(* Schneider Machine Expert - Basic project Pump_Tank_Backup_System_IL, file version 3.0.0.0 *)

HARDWARE
  EthernetConfiguration: SubnetMask=255.255.255.0
  SerialLineConfiguration: Parity=Even, DataBits=8, StopBits=1

SYMBOLS  (address, symbol, comment, settings)
  %TM0      PUMP1_START_DELAY  "Pump 1 Startup Delay - 2 seconds before speed check"  [Type=TON, TimeBase=TimeBase1s, Preset=2]
  %TM1      PUMP2_START_DELAY  "Pump 2 Startup Delay - 2 seconds before speed check"  [Type=TON, TimeBase=TimeBase1s, Preset=2]
  %TM2      PUMP3_START_DELAY  "Pump 3 Startup Delay - 2 seconds before speed check"  [Type=TON, TimeBase=TimeBase1s, Preset=2]
  %I0.0     START_BTN  "System Start Button"
  %I0.1     STOP_BTN  "System Stop Button (NC)"
  %I0.2     E_STOP  "Emergency Stop (NC)"
  %I0.3     PUMP1_SPEED_OK  "Pump 1 Zero Speed Sensor (NC)"
  %I0.4     PUMP2_SPEED_OK  "Pump 2 Zero Speed Sensor (NC)"
  %I0.5     PUMP3_SPEED_OK  "Pump 3 Zero Speed Sensor (NC)"
  %I0.6     TANK1_LOW  "Tank 1 Low Level Switch"
  %I0.7     TANK1_HIGH  "Tank 1 High Level Switch"
  %I0.8     TANK2_LOW  "Tank 2 Low Level Switch"
  %I0.9     TANK2_HIGH  "Tank 2 High Level Switch"
  %I0.10    TANK3_LOW  "Tank 3 Low Level Switch"
  %I0.11    TANK3_HIGH  "Tank 3 High Level Switch"
  %I0.12    PUMP1_OL  "Pump 1 Overload (NC)"
  %I0.13    PUMP2_OL  "Pump 2 Overload (NC)"
  %I0.14    PUMP3_OL  "Pump 3 Overload (NC)"
  %I0.15    FAULT_RESET  "Fault Reset Button"
  %Q0.0     PUMP1_RUN  "Pump 1 Motor Contactor"
  %Q0.1     PUMP2_RUN  "Pump 2 Motor Contactor"
  %Q0.2     PUMP3_RUN  "Pump 3 Motor Contactor"
  %Q0.3     VALVE_12  "Valve Between Tank 1-2"
  %Q0.4     VALVE_23  "Valve Between Tank 2-3"
  %Q0.5     VALVE_13  "Valve Between Tank 1-3"
  %Q0.6     PUMP1_FAULT_IND  "Pump 1 Fault Indicator"
  %Q0.7     PUMP2_FAULT_IND  "Pump 2 Fault Indicator"
  %Q0.8     PUMP3_FAULT_IND  "Pump 3 Fault Indicator"
  %Q0.9     SYSTEM_RUN_IND  "System Running Indicator"
  %Q0.10    ALARM_OUTPUT  "General Alarm Horn"
  %M0       SYSTEM_RUN  "System Running Flag"
  %M1       PUMP1_CMD  "Pump 1 Command"
  %M2       PUMP2_CMD  "Pump 2 Command"
  %M3       PUMP3_CMD  "Pump 3 Command"
  %M10      PUMP1_FAULT  "Pump 1 Fault (Latched)"
  %M11      PUMP2_FAULT  "Pump 2 Fault (Latched)"
  %M12      PUMP3_FAULT  "Pump 3 Fault (Latched)"
  %M20      TANK1_NEEDS_BACKUP  "Tank 1 Backup Mode"
  %M21      TANK2_NEEDS_BACKUP  "Tank 2 Backup Mode"

PouDescriptor Pump_Tank_Backup_IL_Main
  (* PouType=Program *)

// Rung 0: Rung 1
// System Start/Stop with Emergency Stop - Seal-in Circuit
  LD %I0.0                (* START_BTN - Load START button *)
  OR %M0                  (* SYSTEM_RUN - OR with SYSTEM_RUN (seal-in) *)
  ANDN %I0.1              (* STOP_BTN - AND NOT STOP button (NC) *)
  ANDN %I0.2              (* E_STOP - AND NOT E_STOP (NC) *)
  ST %M0                  (* SYSTEM_RUN - Store to SYSTEM_RUN flag *)
  // as ST:
  //   SYSTEM_RUN := (START_BTN OR SYSTEM_RUN) AND NOT STOP_BTN AND NOT E_STOP;

// Rung 1: Rung 2
// Pump 1 Command - Fill Tank 1 when low, stop at high
  LD %M0                  (* SYSTEM_RUN - System running *)
  AND %I0.6               (* TANK1_LOW - AND Tank 1 low level *)
  ANDN %I0.7              (* TANK1_HIGH - AND NOT Tank 1 high level *)
  ANDN %M10               (* PUMP1_FAULT - AND NOT Pump 1 fault *)
  ANDN %I0.12             (* PUMP1_OL - AND NOT Pump 1 overload *)
  ST %M1                  (* PUMP1_CMD - Store to PUMP1_CMD *)
  // as ST:
  //   PUMP1_CMD := SYSTEM_RUN AND TANK1_LOW AND NOT TANK1_HIGH AND NOT PUMP1_FAULT AND NOT PUMP1_OL;

// Rung 2: Rung 3
// Pump 2 Command - Fill Tank 2 when low, stop at high
  LD %M0                  (* SYSTEM_RUN - System running *)
  AND %I0.8               (* TANK2_LOW - AND Tank 2 low level *)
  ANDN %I0.9              (* TANK2_HIGH - AND NOT Tank 2 high level *)
  ANDN %M11               (* PUMP2_FAULT - AND NOT Pump 2 fault *)
  ANDN %I0.13             (* PUMP2_OL - AND NOT Pump 2 overload *)
  ST %M2                  (* PUMP2_CMD - Store to PUMP2_CMD *)
  // as ST:
  //   PUMP2_CMD := SYSTEM_RUN AND TANK2_LOW AND NOT TANK2_HIGH AND NOT PUMP2_FAULT AND NOT PUMP2_OL;

// Rung 3: Rung 4
// Pump 3 Command - Fill Tank 3 when low, stop at high
  LD %M0                  (* SYSTEM_RUN - System running *)
  AND %I0.10              (* TANK3_LOW - AND Tank 3 low level *)
  ANDN %I0.11             (* TANK3_HIGH - AND NOT Tank 3 high level *)
  ANDN %M12               (* PUMP3_FAULT - AND NOT Pump 3 fault *)
  ANDN %I0.14             (* PUMP3_OL - AND NOT Pump 3 overload *)
  ST %M3                  (* PUMP3_CMD - Store to PUMP3_CMD *)
  // as ST:
  //   PUMP3_CMD := SYSTEM_RUN AND TANK3_LOW AND NOT TANK3_HIGH AND NOT PUMP3_FAULT AND NOT PUMP3_OL;

// Rung 4: Rung 5
// Pump 1 Startup Timer and Motor Output
  BLK %TM0                (* PUMP1_START_DELAY - Begin Timer 0 block (PUMP1_START_DELAY) *)
  LD %M1                  (* PUMP1_CMD - Load Pump 1 command *)
  IN                      (* Timer input - starts 2s delay *)
  END_BLK                 (* End timer block *)
  LD %M1                  (* PUMP1_CMD - Load Pump 1 command *)
  ST %Q0.0                (* PUMP1_RUN - Output to PUMP1_RUN contactor *)
  // as ST:
  //   PUMP1_START_DELAY(IN := PUMP1_CMD);
  //   PUMP1_RUN := PUMP1_CMD;

// Rung 5: Rung 6
// Pump 1 Zero Speed Fault - Latching with Reset
  LD %TM0.Q               (* PUMP1_START_DELAY - Timer done (2s elapsed) *)
  ANDN %I0.3              (* PUMP1_SPEED_OK - AND NOT speed OK (zero speed detected) *)
  OR %M10                 (* PUMP1_FAULT - OR with fault latch (seal-in) *)
  ANDN %I0.15             (* FAULT_RESET - AND NOT fault reset button *)
  ST %M10                 (* PUMP1_FAULT - Store to PUMP1_FAULT (latched) *)
  // as ST:
  //   PUMP1_FAULT := (PUMP1_START_DELAY.Q AND NOT PUMP1_SPEED_OK OR PUMP1_FAULT) AND NOT FAULT_RESET;

// Rung 6: Rung 7
// Pump 2 Output - Normal Operation or Backup for Tank 1
  BLK %TM1                (* PUMP2_START_DELAY - Begin Timer 1 block (PUMP2_START_DELAY) *)
  LD %M2                  (* PUMP2_CMD - Load Pump 2 command *)
  OR %M20                 (* TANK1_NEEDS_BACKUP - OR Tank 1 needs backup *)
  IN                      (* Timer input *)
  END_BLK                 (* End timer block *)
  LD %M2                  (* PUMP2_CMD - Load Pump 2 command *)
  OR %M20                 (* TANK1_NEEDS_BACKUP - OR Tank 1 backup mode *)
  ST %Q0.1                (* PUMP2_RUN - Output to PUMP2_RUN contactor *)
  // as ST:
  //   PUMP2_START_DELAY(IN := PUMP2_CMD OR TANK1_NEEDS_BACKUP);
  //   PUMP2_RUN := PUMP2_CMD OR TANK1_NEEDS_BACKUP;

// Rung 7: Rung 8
// Pump 2 Zero Speed Fault Detection
  LD %TM1.Q               (* PUMP2_START_DELAY - Timer done (2s elapsed) *)
  ANDN %I0.4              (* PUMP2_SPEED_OK - AND NOT speed OK (zero speed) *)
  OR %M11                 (* PUMP2_FAULT - OR with fault latch *)
  ANDN %I0.15             (* FAULT_RESET - AND NOT fault reset *)
  ST %M11                 (* PUMP2_FAULT - Store to PUMP2_FAULT *)
  // as ST:
  //   PUMP2_FAULT := (PUMP2_START_DELAY.Q AND NOT PUMP2_SPEED_OK OR PUMP2_FAULT) AND NOT FAULT_RESET;

// Rung 8: Rung 9
// Pump 3 Output - Normal Operation or Backup for Tank 2
  BLK %TM2                (* PUMP3_START_DELAY - Begin Timer 2 block (PUMP3_START_DELAY) *)
  LD %M3                  (* PUMP3_CMD - Load Pump 3 command *)
  OR %M21                 (* TANK2_NEEDS_BACKUP - OR Tank 2 needs backup *)
  IN                      (* Timer input *)
  END_BLK                 (* End timer block *)
  LD %M3                  (* PUMP3_CMD - Load Pump 3 command *)
  OR %M21                 (* TANK2_NEEDS_BACKUP - OR Tank 2 backup mode *)
  ST %Q0.2                (* PUMP3_RUN - Output to PUMP3_RUN contactor *)
  // as ST:
  //   PUMP3_START_DELAY(IN := PUMP3_CMD OR TANK2_NEEDS_BACKUP);
  //   PUMP3_RUN := PUMP3_CMD OR TANK2_NEEDS_BACKUP;

// Rung 9: Rung 10
// Pump 3 Zero Speed Fault Detection
  LD %TM2.Q               (* PUMP3_START_DELAY - Timer done (2s elapsed) *)
  ANDN %I0.5              (* PUMP3_SPEED_OK - AND NOT speed OK *)
  OR %M12                 (* PUMP3_FAULT - OR with fault latch *)
  ANDN %I0.15             (* FAULT_RESET - AND NOT fault reset *)
  ST %M12                 (* PUMP3_FAULT - Store to PUMP3_FAULT *)
  // as ST:
  //   PUMP3_FAULT := (PUMP3_START_DELAY.Q AND NOT PUMP3_SPEED_OK OR PUMP3_FAULT) AND NOT FAULT_RESET;

// Rung 10: Rung 11
// Tank 1 Backup Request - Pump 2 takes over when Pump 1 fails
  LD %M10                 (* PUMP1_FAULT - Pump 1 fault active *)
  AND %I0.6               (* TANK1_LOW - AND Tank 1 low level *)
  ANDN %I0.7              (* TANK1_HIGH - AND NOT Tank 1 high *)
  ANDN %M11               (* PUMP2_FAULT - AND NOT Pump 2 fault (backup available) *)
  ST %M20                 (* TANK1_NEEDS_BACKUP - Store to TANK1_NEEDS_BACKUP *)
  // as ST:
  //   TANK1_NEEDS_BACKUP := PUMP1_FAULT AND TANK1_LOW AND NOT TANK1_HIGH AND NOT PUMP2_FAULT;

// Rung 11: Rung 12
// Tank 2 Backup Request - Pump 3 takes over when Pump 2 fails
  LD %M11                 (* PUMP2_FAULT - Pump 2 fault active *)
  AND %I0.8               (* TANK2_LOW - AND Tank 2 low level *)
  ANDN %I0.9              (* TANK2_HIGH - AND NOT Tank 2 high *)
  ANDN %M12               (* PUMP3_FAULT - AND NOT Pump 3 fault (backup available) *)
  ST %M21                 (* TANK2_NEEDS_BACKUP - Store to TANK2_NEEDS_BACKUP *)
  // as ST:
  //   TANK2_NEEDS_BACKUP := PUMP2_FAULT AND TANK2_LOW AND NOT TANK2_HIGH AND NOT PUMP3_FAULT;

// Rung 12: Rung 13
// Valve 1-2 Opens when Tank 1 in Backup Mode
  LD %M20                 (* TANK1_NEEDS_BACKUP - Tank 1 needs backup *)
  ST %Q0.3                (* VALVE_12 - Open VALVE_12 (between Tank 1 and 2) *)
  // as ST:
  //   VALVE_12 := TANK1_NEEDS_BACKUP;

// Rung 13: Rung 14
// Valve 2-3 Opens when Tank 2 in Backup Mode
  LD %M21                 (* TANK2_NEEDS_BACKUP - Tank 2 needs backup *)
  ST %Q0.4                (* VALVE_23 - Open VALVE_23 (between Tank 2 and 3) *)
  // as ST:
  //   VALVE_23 := TANK2_NEEDS_BACKUP;

// Rung 14: Rung 15
// Pump 1 Fault Indicator Light
  LD %M10                 (* PUMP1_FAULT - Pump 1 fault *)
  ST %Q0.6                (* PUMP1_FAULT_IND - PUMP1_FAULT_IND light *)
  // as ST:
  //   PUMP1_FAULT_IND := PUMP1_FAULT;

// Rung 15: Rung 16
// Pump 2 Fault Indicator Light
  LD %M11                 (* PUMP2_FAULT - Pump 2 fault *)
  ST %Q0.7                (* PUMP2_FAULT_IND - PUMP2_FAULT_IND light *)
  // as ST:
  //   PUMP2_FAULT_IND := PUMP2_FAULT;

// Rung 16: Rung 17
// Pump 3 Fault Indicator Light
  LD %M12                 (* PUMP3_FAULT - Pump 3 fault *)
  ST %Q0.8                (* PUMP3_FAULT_IND - PUMP3_FAULT_IND light *)
  // as ST:
  //   PUMP3_FAULT_IND := PUMP3_FAULT;

// Rung 17: Rung 18
// System Running Indicator Light
  LD %M0                  (* SYSTEM_RUN - System running *)
  ST %Q0.9                (* SYSTEM_RUN_IND - SYSTEM_RUN_IND light *)
  // as ST:
  //   SYSTEM_RUN_IND := SYSTEM_RUN;

// Rung 18: Rung 19
// General Alarm - Any Pump Fault Activates Horn
  LD %M10                 (* PUMP1_FAULT - Pump 1 fault *)
  OR %M11                 (* PUMP2_FAULT - OR Pump 2 fault *)
  OR %M12                 (* PUMP3_FAULT - OR Pump 3 fault *)
  ST %Q0.10               (* ALARM_OUTPUT - ALARM_OUTPUT horn *)
  // as ST:
  //   ALARM_OUTPUT := PUMP1_FAULT OR PUMP2_FAULT OR PUMP3_FAULT;
